(* CoDeSys 2.3.9.35 project: ACIONAMENTO.pro *)
(* Author: Hemerson *)
(* Libraries: SysLibTargetVisu.lib 26.11.08 09:50:36, Standard.lib 26.11.08 09:46:20, Iecsfc.lib 26.11.08 09:46:14, DU35x.lib 7.7.11 15:59:53, SYSLIBCALLBACK.LIB 26.11.08 09:50:38 *)

(* PLC configuration (modules and I/O channels)
Communication [Comunica] node 0, in %IB0 out %QB0
  COM1 [COM1] node 0, in %IB0 out %QB0 {BaudRate = 115200; Paridade = No Parity; StopBits = 1 Stop Bit; Modem = Without RTS/CTS; Delay = 5}
    MToolIEC [Codesys] node 0, in %IB0 out %QB0
  COM2 [COM2] node 1, in %IB0 out %QB0 {BaudRate = 115200; Paridade = No Parity; StopBits = 1 Stop Bit; Modem = Without RTS/CTS; Delay = 5}
    Disable [Desabilitado485] node 0, in %IB0 out %QB0
Digital Inputs 0 [Entradas0] node 0, in %IW0 out %QB0
  I00 AT %IX0.0 [BitInput] I0.0
  I01 AT %IX0.1 [BitInput] I0.1
  I02 AT %IX0.2 [BitInput] I0.2
  I03 AT %IX0.3 [BitInput] I0.3
  I04 AT %IX0.4 [BitInput] I0.4
  I05 AT %IX0.5 [BitInput] I0.5
  I06 AT %IX0.6 [BitInput] I0.6
  I07 AT %IX0.7 [BitInput] I0.7
  I08 AT %IX0.8 [BitInput] I0.8
Digital Inputs 1 [Entradas1] node 0, in %IW1 out %QB0
  I10 AT %IX1.0 [BitInput] I1.0
  I11 AT %IX1.1 [BitInput] I1.1
  I12 AT %IX1.2 [BitInput] I1.2
  I13 AT %IX1.3 [BitInput] I1.3
  I14 AT %IX1.4 [BitInput] I1.4
  I15 AT %IX1.5 [BitInput] I1.5
  I16 AT %IX1.6 [BitInput] I1.6
  I17 AT %IX1.7 [BitInput] I1.7
  I18 AT %IX1.8 [BitInput] I1.8
Digital Inputs 2 [Entradas2] node 0, in %IW2 out %QB0
  I20 AT %IX2.0 [BitInput] I2.0
  I21 AT %IX2.1 [BitInput] I2.1
AI0 AT %IW4 [WordInput] AI0 {TipoAnalogica = Channel Disable; FiltroAnalogica = Filter 0 - AI=2ms  / AV=90ms; FundoEscala = 0}
AI1 AT %IW5 [WordInput] AI1 {TipoAnalogica = Channel Disable; FiltroAnalogica = Filter 0 - AI=2ms  / AV=90ms; FundoEscala = 0}
AI2 AT %IW6 [WordInput] AI2 {TipoAnalogica = Channel Disable; FiltroAnalogica = Filter 0 - AI=2ms  / AV=90ms; FundoEscala = 0}
AI3 AT %IW7 [WordInput] AI3 {TipoAnalogica = Channel Disable; FiltroAnalogica = Filter 0 - AI=2ms  / AV=90ms; FundoEscala = 0}
Fast Inputs [EntradasRapidas] node 1, in %IB16 out %QB0
  Block 0 [Bloco0] node 0, in %IB16 out %QB0
    Disable [DesabilitadoBloco0] node 0, in %IB16 out %QB0
  Block 1 [Bloco1] node 1, in %IB16 out %QB0
    Disable [DesabilitadoBloco1] node 0, in %IB16 out %QB0
  Configurable Input Block 0 [EntradaConfiBloco0] node 2, in %IB16 out %QB0
    Counter 0 [EntradaConfContador0] node 0, in %IB16 out %QB0 {EntradaConfiguravelContador = Disable}
  Configurable Input Block 1 [EntradaConfiBloco1] node 3, in %IB16 out %QB0
    Counter 2 [EntradaConfContador2] node 0, in %IB16 out %QB0 {EntradaConfiguravelContador = Disable}
Outputs [Saidas] node 1, in %IB13 out %QB0
  Digital Outputs 0 [Saidas0] node 0, in %IW0 out %QW0
    Q00 AT %QX0.0 [BitOutput] Q0.0
    Q01 AT %QX0.1 [BitOutput] Q0.1
    Q02 AT %QX0.2 [BitOutput] Q0.2
    Q03 AT %QX0.3 [BitOutput] Q0.3
    Q04 AT %QX0.4 [BitOutput] Q0.4
    Q05 AT %QX0.5 [BitOutput] Q0.5
    Q06 AT %QX0.6 [BitOutput] Q0.6
    Q07 AT %QX0.7 [BitOutput] Q0.7
  Digital Outputs 1 [Saidas1] node 0, in %IW0 out %QW1
    Q10 AT %QX1.0 [BitOutput] Q1.0
    Q11 AT %QX1.1 [BitOutput] Q1.1
    Q12 AT %QX1.2 [BitOutput] Q1.2
    Q13 AT %QX1.3 [BitOutput] Q1.3
    Q14 AT %QX1.4 [BitOutput] Q1.4
    Q15 AT %QX1.5 [BitOutput] Q1.5
    Q16 AT %QX1.6 [BitOutput] Q1.6
    Q17 AT %QX1.7 [BitOutput] Q1.7
  Analog Outputs [SaidaAnalogica] node 0, in %IW0 out %QW3
    AO0 AT %QW3 [WordOutput] AO0 {TipoAnalogica = Channel Disable; FundoEscala = 0}
    AO1 AT %QW4 [WordOutput] AO1 {TipoAnalogica = Channel Disable; FundoEscala = 0}
  Fast Outputs [SaidasRapidas] node 1, in %IB0 out %QB10
    Fast Output 0 Disable [DesabilitadoF0] node 0, in %IB0 out %QB10
    Fast Output 1 Disable [DesabilitadoF1] node 1, in %IB0 out %QB10
  Counter Output [SaidasContador] node 2, in %IB0 out %QB10
    Block 0 Output Disable [DesabilitadoSaidaBloco0] node 0, in %IB0 out %QB10
    Block 1 Output Disable [DesabilitadoSaidaBloco1] node 1, in %IB0 out %QB10
External Events [Eventos] node 2, in %IB13 out %QB6
  Timer Event [TimerEvent] node 0, in %IB13 out %QB6 {Intervalo = 10}
*)

(* Global variable list: Variáveis globais *)
VAR_GLOBAL
	D  AT %IX0.0: BOOL;
	A1 AT %IX0.1: BOOL;
	A2 AT %IX0.2: BOOL;
	A3 AT %IX0.3: BOOL;
	A4 AT %IX0.4: BOOL;
	A5 AT %IX0.5: BOOL;
	A6 AT %IX0.6: BOOL;

	M1 AT %QX1.0: BOOL;
	M2 AT %QX1.1: BOOL;
	M3 AT %QX1.2: BOOL;
	M4 AT %QX1.3: BOOL;
	M5 AT %QX1.4: BOOL;
	M6 AT %QX1.5: BOOL;
	TEMP1: TON;
	TEMP2: TON;
	TEMP3: TON;
	M: BOOL;
	TEMP: TON;
	TEMP4: TON;
	TEMP5: TON;
	TEMP6: TON;
END_VAR

(* POU PLC_PRG, LD *)
PROGRAM PLC_PRG
VAR
	D  AT %IX0.0: BOOL;
	A1 AT %IX0.1: BOOL;
	A2 AT %IX0.2: BOOL;
	A3 AT %IX0.3: BOOL;
	A4 AT %IX0.4: BOOL;
	A5 AT %IX0.5: BOOL;
	A6 AT %IX0.6: BOOL;

	M1 AT %QX1.0: BOOL;
	M2 AT %QX1.1: BOOL;
	M3 AT %QX1.2: BOOL;
	M4 AT %QX1.3: BOOL;
	M5 AT %QX1.4: BOOL;
	M6 AT %QX1.5: BOOL;
	TEMP1: TON;
	TEMP2: TON;
	TEMP3: TON;
	M: BOOL;
	TEMP: TON;
	TEMP4: TON;
	TEMP5: TON;
	TEMP6: TON;
END_VAR
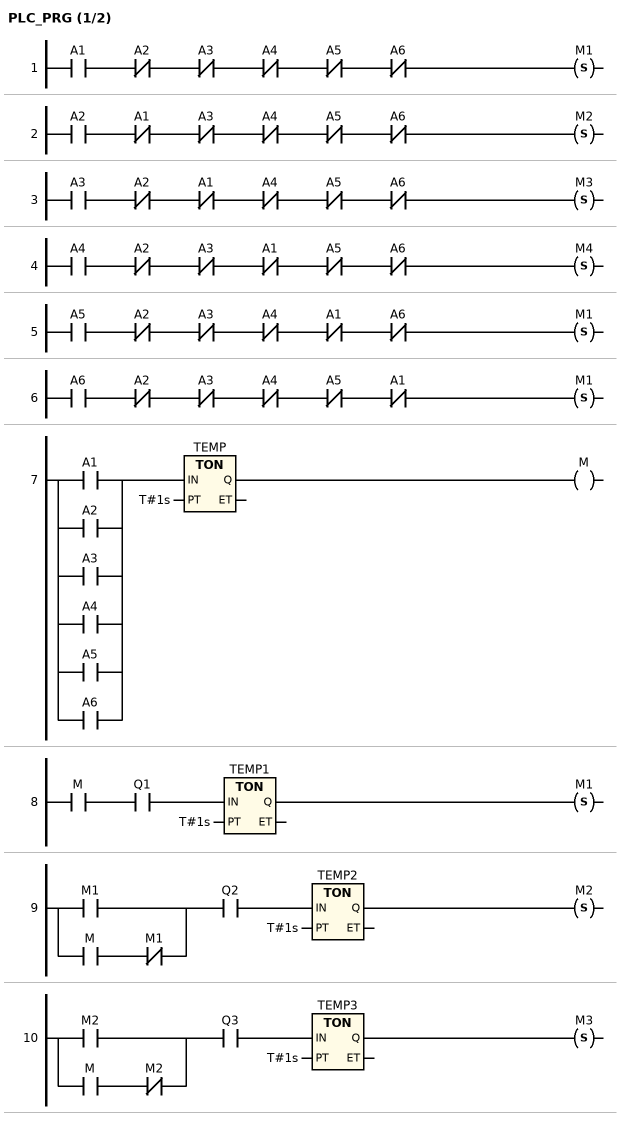
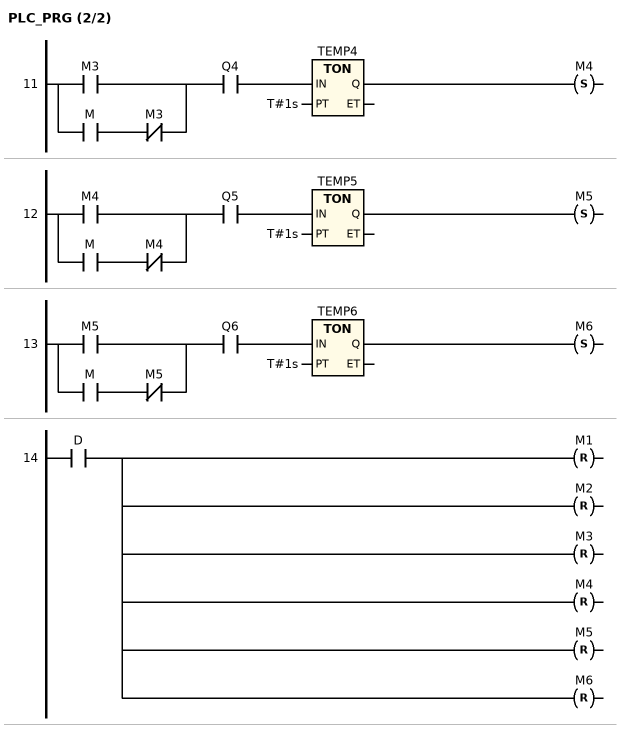
_LD_ (* Ladder Diagram *)
NETWORK 1
	[A1] - [/A2] - [/A3] - [/A4] - [/A5] - [/A6] --- (S M1)
NETWORK 2
	[A2] - [/A1] - [/A3] - [/A4] - [/A5] - [/A6] --- (S M2)
NETWORK 3
	[A3] - [/A2] - [/A1] - [/A4] - [/A5] - [/A6] --- (S M3)
NETWORK 4
	[A4] - [/A2] - [/A3] - [/A1] - [/A5] - [/A6] --- (S M4)
NETWORK 5
	[A5] - [/A2] - [/A3] - [/A4] - [/A1] - [/A6] --- (S M1)
NETWORK 6
	[A6] - [/A2] - [/A3] - [/A4] - [/A5] - [/A1] --- (S M1)
NETWORK 7
	{ [A1] | [A2] | [A3] | [A4] | [A5] | [A6] } - TEMP:TON(IN: *, PT: T#1s) --- (M)
NETWORK 8
	[M] - [Q1] - TEMP1:TON(IN: *, PT: T#1s) --- (S M1)
NETWORK 9
	{ [M1] | [M] - [/M1] } - [Q2] - TEMP2:TON(IN: *, PT: T#1s) --- (S M2)
NETWORK 10
	{ [M2] | [M] - [/M2] } - [Q3] - TEMP3:TON(IN: *, PT: T#1s) --- (S M3)
NETWORK 11
	{ [M3] | [M] - [/M3] } - [Q4] - TEMP4:TON(IN: *, PT: T#1s) --- (S M4)
NETWORK 12
	{ [M4] | [M] - [/M4] } - [Q5] - TEMP5:TON(IN: *, PT: T#1s) --- (S M5)
NETWORK 13
	{ [M5] | [M] - [/M5] } - [Q6] - TEMP6:TON(IN: *, PT: T#1s) --- (S M6)
NETWORK 14
	[D] --- (R M1) (R M2) (R M3) (R M4) (R M5) (R M6)
_END_LD_
(* the same logic as Structured Text *)
(* Network 1 *)
IF A1 AND NOT A2 AND NOT A3 AND NOT A4 AND NOT A5 AND NOT A6 THEN M1 := TRUE; END_IF;
(* Network 2 *)
IF A2 AND NOT A1 AND NOT A3 AND NOT A4 AND NOT A5 AND NOT A6 THEN M2 := TRUE; END_IF;
(* Network 3 *)
IF A3 AND NOT A2 AND NOT A1 AND NOT A4 AND NOT A5 AND NOT A6 THEN M3 := TRUE; END_IF;
(* Network 4 *)
IF A4 AND NOT A2 AND NOT A3 AND NOT A1 AND NOT A5 AND NOT A6 THEN M4 := TRUE; END_IF;
(* Network 5 *)
IF A5 AND NOT A2 AND NOT A3 AND NOT A4 AND NOT A1 AND NOT A6 THEN M1 := TRUE; END_IF;
(* Network 6 *)
IF A6 AND NOT A2 AND NOT A3 AND NOT A4 AND NOT A5 AND NOT A1 THEN M1 := TRUE; END_IF;
(* Network 7 *)
TEMP(IN := A1 OR A2 OR A3 OR A4 OR A5 OR A6, PT := T#1s);
M := TEMP.Q;
(* Network 8 *)
TEMP1(IN := M AND Q1, PT := T#1s);
IF TEMP1.Q THEN M1 := TRUE; END_IF;
(* Network 9 *)
TEMP2(IN := (M1 OR M AND NOT M1) AND Q2, PT := T#1s);
IF TEMP2.Q THEN M2 := TRUE; END_IF;
(* Network 10 *)
TEMP3(IN := (M2 OR M AND NOT M2) AND Q3, PT := T#1s);
IF TEMP3.Q THEN M3 := TRUE; END_IF;
(* Network 11 *)
TEMP4(IN := (M3 OR M AND NOT M3) AND Q4, PT := T#1s);
IF TEMP4.Q THEN M4 := TRUE; END_IF;
(* Network 12 *)
TEMP5(IN := (M4 OR M AND NOT M4) AND Q5, PT := T#1s);
IF TEMP5.Q THEN M5 := TRUE; END_IF;
(* Network 13 *)
TEMP6(IN := (M5 OR M AND NOT M5) AND Q6, PT := T#1s);
IF TEMP6.Q THEN M6 := TRUE; END_IF;
(* Network 14 *)
IF D THEN M1 := FALSE; M2 := FALSE; M3 := FALSE; M4 := FALSE; M5 := FALSE; M6 := FALSE; END_IF;
END_PROGRAM

(* Visualisation main
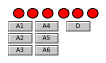
ellipse at (9,8)-(20,18): alarm colour if PLC_PRG.M1
ellipse at (23,8)-(34,18): alarm colour if .M2
ellipse at (38,8)-(49,18): alarm colour if .M3
button at (4,21)-(28,31): text "A1"; toggles PLC_PRG.A1
button at (4,33)-(28,43): text "A2"; toggles PLC_PRG.A2
button at (4,45)-(28,55): text "A3"; toggles PLC_PRG.A3
button at (31,21)-(54,31): text "A4"; toggles PLC_PRG.A4
button at (31,33)-(54,43): text "A5"; toggles PLC_PRG.A5
button at (31,45)-(54,55): text "A6"; toggles PLC_PRG.A6
button at (62,21)-(86,31): text "D"; toggles PLC_PRG.D
ellipse at (54,8)-(65,18): alarm colour if PLC_PRG.M4
ellipse at (68,8)-(79,18): alarm colour if PLC_PRG.M5
ellipse at (83,8)-(94,18): alarm colour if PLC_PRG.M6
*)
